{attribute 'GeneratedUsingTerminal: EP6224-2022-0016'}
{attribute addProperty BoxType "EP6224-2022-0016"}
{attribute addProperty Id "DeviceState_Inputs_DeviceAT %I*DeviceState_Inputs_Device_A12105982DeviceState_InputsAT %I*DeviceState_Inputs_4751FF764IO_Inputs_Channel_1EMPTY_STRUCTURE0IO_Inputs_Channel_2EMPTY_STRUCTURE0IO_Inputs_Channel_3EMPTY_STRUCTURE0IO_Inputs_Channel_4EMPTY_STRUCTURE0IO_Outputs_Channel_1EMPTY_STRUCTURE0IO_Outputs_Channel_2EMPTY_STRUCTURE0IO_Outputs_Channel_3EMPTY_STRUCTURE0IO_Outputs_Channel_4EMPTY_STRUCTURE0WcStateAT %I*WcState_9091E0EB2InfoDataAT %I*InfoData_41C547A32"}
{attribute addProperty CRC "191202523"}
{attribute addProperty Size "10"}
TYPE EP6224_0B6584DB EXTENDS EtcSlaveTerminalBase_947E5A46 :
STRUCT
	{attribute addProperty Name "DeviceState_Inputs_Device"}
	DeviceState_Inputs_Device : DeviceState_Inputs_Device_A1210598;
	{attribute addProperty Name "DeviceState_Inputs"}
	DeviceState_Inputs : DeviceState_Inputs_4751FF76;
	{attribute addProperty Name "IO_Inputs_Channel_1"}
	IO_Inputs_Channel_1 : EMPTY_STRUCTURE;
	{attribute addProperty Name "IO_Inputs_Channel_2"}
	IO_Inputs_Channel_2 : EMPTY_STRUCTURE;
	{attribute addProperty Name "IO_Inputs_Channel_3"}
	IO_Inputs_Channel_3 : EMPTY_STRUCTURE;
	{attribute addProperty Name "IO_Inputs_Channel_4"}
	IO_Inputs_Channel_4 : EMPTY_STRUCTURE;
	{attribute addProperty Name "IO_Outputs_Channel_1"}
	IO_Outputs_Channel_1 : EMPTY_STRUCTURE;
	{attribute addProperty Name "IO_Outputs_Channel_2"}
	IO_Outputs_Channel_2 : EMPTY_STRUCTURE;
	{attribute addProperty Name "IO_Outputs_Channel_3"}
	IO_Outputs_Channel_3 : EMPTY_STRUCTURE;
	{attribute addProperty Name "IO_Outputs_Channel_4"}
	IO_Outputs_Channel_4 : EMPTY_STRUCTURE;
	{attribute addProperty Name "WcState"}
	WcState : WcState_9091E0EB;
	{attribute addProperty Name "InfoData"}
	InfoData : InfoData_41C547A3;
END_STRUCT
END_TYPE

(* stored: Version 1.2.0.0, ProductVersion 3.1.4024.9
   DUT EP6224_0B6584DB: Id {4299d923-83e2-4789-be46-4a0278e725c6} *)
